Staubli VAL3: setLastError.pgx

program setLastError(num x_nError)
begin

  nLastError=x_nError

end
